FUNCTION_BLOCK FB_GrandChild EXTENDS FB_Child2
VAR_INPUT
END_VAR
VAR_OUTPUT
END_VAR
VAR
END_VAR

END_FUNCTION_BLOCK

(* stored: Version 1.1.0.1, ProductVersion 3.1.4024.16
   POU FB_GrandChild: Id {80c841bc-6f42-4054-82b0-4d59ce163ecd}, SpecialFunc None *)
